FUNCTION_BLOCK FB_ManualStateMachine
VAR_INPUT
	startCycle 			: BOOL;
	continueToTop		: BOOL;
	continueToBottom	: BOOL;
	endAtTop			: BOOL;
	endAtBottom			: BOOL;
END_VAR
VAR_OUTPUT
	moveBottom			: BOOL;
	moveTop				: BOOL;
END_VAR
VAR
END_VAR

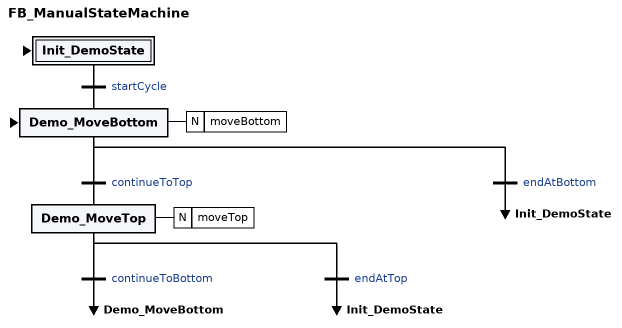
INITIAL_STEP Init_DemoState:
END_STEP
TRANSITION FROM Init_DemoState TO Demo_MoveBottom
    := startCycle;
END_TRANSITION
STEP Demo_MoveBottom:
    moveBottom(N);
END_STEP
TRANSITION FROM Demo_MoveBottom TO Demo_MoveTop
    := continueToTop;
END_TRANSITION
TRANSITION FROM Demo_MoveBottom TO Init_DemoState
    := endAtBottom;
END_TRANSITION
STEP Demo_MoveTop:
    moveTop(N);
END_STEP
TRANSITION FROM Demo_MoveTop TO Demo_MoveBottom
    := continueToBottom;
END_TRANSITION
TRANSITION FROM Demo_MoveTop TO Init_DemoState
    := endAtTop;
END_TRANSITION
// branch label Branch0_DemoState

END_FUNCTION_BLOCK

(* stored: Version 1.1.0.1, ProductVersion 3.1.4024.12
   POU FB_ManualStateMachine: Id {90634356-0d72-4b86-a14c-3dcf81e6168f}, SpecialFunc None *)
